FUNCTION_BLOCK AR_MULTIME (* Multiplies time value with numerical values *)
  (* Standard: 61131-3; Classification: standard arithmetic function; Description: Copyright (c) 2013 TU Wien ACIN This program and the accompanying materials are made available under the terms of the Eclipse Public License 2.0 which is available at https://www.eclipse.org/legal/epl-2.0/ SPDX-License-Identifier: EPL-2.0 *)
  (* Version 3.0, 2025-04-14, Patrick Aigner, changed package *)
  (* Version 1.0, 2013-09-12, Monika Wenger, TU Wien ACIN *)
  PACKAGE adapter::iec61131::arithmetic;
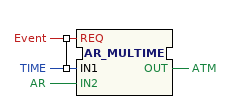
  EVENT_INPUT
    REQ WITH IN1; (* Normal Execution Request *)
  END_EVENT
  VAR_INPUT
    IN1 : TIME; (* First function input *)
  END_VAR
  SOCKETS
    IN2 : adapter::types::unidirectional::AR; (* Second function input *)
  END_SOCKETS
  PLUGS
    OUT : adapter::types::unidirectional::ATM; (* IN1 multiplied by IN2 *)
  END_PLUGS
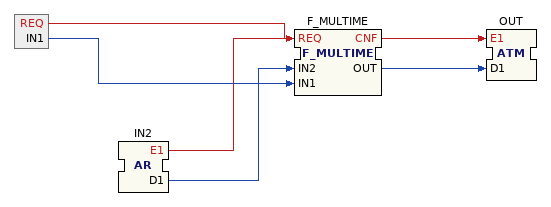
  FBS
    F_MULTIME : iec61131::arithmetic::F_MULTIME;
  END_FBS
  EVENT_CONNECTIONS
    F_MULTIME.CNF TO OUT.E1;
    IN2.E1 TO F_MULTIME.REQ;
    REQ TO F_MULTIME.REQ;
  END_CONNECTIONS
  DATA_CONNECTIONS
    F_MULTIME.OUT TO OUT.D1;
    IN2.D1 TO F_MULTIME.IN2;
    IN1 TO F_MULTIME.IN1;
  END_CONNECTIONS
END_FUNCTION_BLOCK
